INTERFACE I_SERIALCONTROLLER

PROPERTY Suffix : STRING(15)
SET
END_SET
GET
END_GET
END_PROPERTY

PROPERTY Prefix : STRING(15)
GET
END_GET
SET
END_SET
END_PROPERTY

METHOD Receive : DINT
VAR_INPUT
	ptr_data : PVOID;
END_VAR
END_METHOD

METHOD FastBackgroundTask : DINT
VAR_INPUT
END_VAR
END_METHOD

METHOD Send : DINT
VAR_INPUT
	ptr_data : PVOID;
	length : UDINT;
END_VAR
END_METHOD

PROPERTY TimeOut : TIME
SET
END_SET
GET
END_GET
END_PROPERTY

END_INTERFACE

(* stored: Version 1.1.0.1, ProductVersion 3.1.4019.2
   Itf I_SERIALCONTROLLER: Id {9bbed68e-90bf-49b5-80e8-9936eebff057}
   Property Suffix: Id {09030867-e34c-40f1-b43f-6915fa0afcb6}
   Set Set: Id {e4bda62d-94c4-40b3-8cf6-515e0c536fdf}
   Get Get: Id {e752c183-4227-4750-af91-c1507e574ce5}
   Property Prefix: Id {239b2626-0c6d-479e-882b-e5a3cdc2b253}
   Get Get: Id {08947e29-061f-48b5-b0d2-74e830210b30}
   Set Set: Id {f987d17b-f6d6-4c58-ac1b-797a89ea39f1}
   Method Receive: Id {59d14c9f-5b9d-4a12-8fd7-387828c2f26a}
   Method FastBackgroundTask: Id {9bd29ca8-93f1-4106-bc79-680baa339010}
   Method Send: Id {b0fdd19f-179e-45f8-8286-92cd1bcce424}
   Property TimeOut: Id {e1dba4e4-9910-4d37-af28-9b2defa3732b}
   Set Set: Id {307b1541-1357-4b41-81d4-e3799c735d1a}
   Get Get: Id {bb55c62b-a80a-4d92-aad3-2248262c986c} *)
